# EPICS substitutions: LVREMOTE/LVREMOTE-IOC-01App/Db/lvremote_dds_tensile_stress_rig.substitutions
file lvremote_header.template {
    pattern { RECSIM, DISABLE }
    { "\$(RECSIM)", "\$(DISABLE)", }
}

file  lvremote_binary.template {
  pattern
    {DEVICE, P, NAME, IND, CONTROL, ZERO, ONE, VI, PORT, READONLY, DESCRIPTION, SCAN, HIGH}

    {"DDS_STRESS_RIG", "\$(P)", "ULIMIT:ENABLED", "EnableUL", "EnableUL", "False", "True", "C:/Instrument/Dev/ibex_vis/Drivers/DDS/dds Server.vi", "\$(NUM_PORT)", "", "Enable Upper Limit", "1 second", ""}
    {"DDS_STRESS_RIG", "\$(P)", "LLIMIT:ENABLED", "EnableLL", "EnableLL", "False", "True", "C:/Instrument/Dev/ibex_vis/Drivers/DDS/dds Server.vi", "\$(NUM_PORT)", "", "Enable Lower Limit", "1 second", ""}
    {"DDS_STRESS_RIG", "\$(P)", "SPEED:SET", "SetSpeed", "SetSpeed", "False", "True", "C:/Instrument/Dev/ibex_vis/Drivers/DDS/dds Server.vi", "\$(NUM_PORT)", "", "Set Speed", "1 second", "0.1"},
    {"DDS_STRESS_RIG", "\$(P)", "READ:START", "StartRead", "StartRead", "False", "True", "C:/Instrument/Dev/ibex_vis/Drivers/DDS/dds Server.vi", "\$(NUM_PORT)", "", "Start Reading", "1 second", "0.1"},
    {"DDS_STRESS_RIG", "\$(P)", "READ:STOP", "StopRead", "StopRead", "False", "True", "C:/Instrument/Dev/ibex_vis/Drivers/DDS/dds Server.vi", "\$(NUM_PORT)", "", "Stop Reading", "1 second", "0.1"},
    {"DDS_STRESS_RIG", "\$(P)", "MEAS:START", "StartMeasurement", "StartMeasurement", "False", "True", "C:/Instrument/Dev/ibex_vis/Drivers/DDS/dds Server.vi", "\$(NUM_PORT)", "", "Start Measurement", "1 second", "0.1"},
    {"DDS_STRESS_RIG", "\$(P)", "MEAS:STOP", "StopMeasurement", "StopMeasurement", "False", "True", "C:/Instrument/Dev/ibex_vis/Drivers/DDS/dds Server.vi", "\$(NUM_PORT)", "", "Stop Measurement", "1 second", "0.1"},
    {"DDS_STRESS_RIG", "\$(P)", "MOT:START", "StartMotor", "StartMotor", "False", "True", "C:/Instrument/Dev/ibex_vis/Drivers/DDS/dds Server.vi", "\$(NUM_PORT)", "", "Start Motor", "1 second", "0.1"},
    {"DDS_STRESS_RIG", "\$(P)", "MOT:STOP", "StopMotor", "StopMotor", "False", "True", "C:/Instrument/Dev/ibex_vis/Drivers/DDS/dds Server.vi", "\$(NUM_PORT)", "", "Stop Motor", "1 second", "0.1"}
}

file  lvremote_double.template {
  pattern
    {DEVICE, P, NAME, IND, CONTROL, VI, PORT, READONLY, WRITEONLY, SIMRECORD, DESCRIPTION, SCAN}

    {"DDS_STRESS_RIG", "\$(P)", "_SPEED", "Speed", "Speed", "C:/Instrument/Dev/ibex_vis/Drivers/DDS/dds Server.vi", "\$(NUM_PORT)", "","","", "Speed", "1 second"},
    {"DDS_STRESS_RIG", "\$(P)", "UPPER_LIMIT", "Upper Limit", "Upper Limit", "C:/Instrument/Dev/ibex_vis/Drivers/DDS/dds Server.vi", "\$(NUM_PORT)", "","","", "Upper Limit", "1 second"},
    {"DDS_STRESS_RIG", "\$(P)", "LOWER_LIMIT", "Lower Limit", "Lower Limit", "C:/Instrument/Dev/ibex_vis/Drivers/DDS/dds Server.vi", "\$(NUM_PORT)", "","","", "Lower Limit", "1 second"}
}

file  lvremote_enum.template {
  pattern
    {DEVICE, P, NAME, IND, CONTROL, VI, PORT, PORT2, READONLY, DESCRIPTION, SCAN, ZRST, ONST, TWST, THST,FRST,FVST,SXST, ZRVL, ONVL, TWVL, THVL,FRVL,FVVL,SXVL}

    {"DDS_STRESS_RIG", "\$(P)", "MODE:SPEED", "Mode", "Mode", "C:/Instrument/Dev/ibex_vis/Drivers/DDS/dds Server.vi", "\$(NUM_PORT)", "\$(STRING_PORT)", "", "Speed Mode", "1 second", "Manual", "Standard", "Load Const", "","","","", "0", "1", "2", "0","0","0","0"},
    {"DDS_STRESS_RIG", "\$(P)", "CONTROL:SPEED", "Control", "Control", "C:/Instrument/Dev/ibex_vis/Drivers/DDS/dds Server.vi", "\$(NUM_PORT)", "\$(STRING_PORT)", "", "Speed Control", "1 second", "Tacho", "Load", "Elongation", "Elongation 2","","","", "0", "1", "2", "3","0","0","0"},
    {"DDS_STRESS_RIG", "\$(P)", "DIRECTION:SPEED", "Direction", "Direction", "C:/Instrument/Dev/ibex_vis/Drivers/DDS/dds Server.vi", "\$(NUM_PORT)", "\$(STRING_PORT)", "", "Speed Direction", "1 second", "Forward", "Forward2", "Reverse", "","","","", "0", "1", "2", "3","0","0","0"},
    {"DDS_STRESS_RIG", "\$(P)", "MODE:STAT", "Mode String", "Set Mode", "C:/Instrument/Dev/ibex_vis/Drivers/DDS/dds Server.vi", "\$(NUM_PORT)", "\$(STRING_PORT)", "", "Set Mode", "1 second", "Manual", "Standard", "Load Const", "Elong 2","","","", "0", "1", "2", "3","0","0","0"},
    {"DDS_STRESS_RIG", "\$(P)", "MOT:MODE", "Motor Control Mode String", "Set Control", "C:/Instrument/Dev/ibex_vis/Drivers/DDS/dds Server.vi", "\$(NUM_PORT)", "\$(STRING_PORT)", "", "Set Control", "1 second", "Tacho", "Load", "Elongation", "Elongation 2","","","", "0", "1", "2", "3","0","0","0"},
    {"DDS_STRESS_RIG", "\$(P)", "DIR", "Direction String", "Set Direction", "C:/Instrument/Dev/ibex_vis/Drivers/DDS/dds Server.vi", "\$(NUM_PORT)", "\$(STRING_PORT)", "", "Set Direction", "1 second", "Forward", "Forward2", "Reverse", "","","","", "0", "1", "2", "3","0","0","0"},
    {"DDS_STRESS_RIG", "\$(P)", "CHANNEL", "Choose Channel", "Choose Channel", "C:/Instrument/Dev/ibex_vis/Drivers/DDS/dds Server.vi", "\$(NUM_PORT)", "\$(STRING_PORT)", "", "Channel", "1 second", "Time", "Load", "Elongation", "Elong2","","","", "0", "1", "2", "3","0","0","0"}

    {"DDS_STRESS_RIG", "\$(P)", "MOT:STAT", "Motor Status String", "Motor Status String", "C:/Instrument/Dev/ibex_vis/Drivers/DDS/dds Server.vi", "\$(NUM_PORT)", "\$(STRING_PORT)", "#", "Motor Status", "1 second", "Stop", "Forward", "Reverse", "","","","", "0", "1", "2", "0","0","0","0"},
    {"DDS_STRESS_RIG", "\$(P)", "CON:STAT", "Control Status String", "Control Status String", "C:/Instrument/Dev/ibex_vis/Drivers/DDS/dds Server.vi", "\$(NUM_PORT)", "\$(STRING_PORT)", "#", "Control Status", "1 second", "Idle", "Read", "Active","Hold","HoldEnd","AutoZero","AutoKeepConst", "0","1","2","3","4","5","6"},
    {"DDS_STRESS_RIG", "\$(P)", "TEMP:STAT", "Temp Status String", "Temp Status String", "C:/Instrument/Dev/ibex_vis/Drivers/DDS/dds Server.vi", "\$(NUM_PORT)", "\$(STRING_PORT)", "#", "Temp Status String", "1 second", "Stop", "Heating", "Cooling", "","","","", "0", "1", "2", "0","0","0","0"},
}

file lvremote_array.template {
  pattern
  {DEVICE, P, NAME, IND, CONTROL, VI, PORT, DESCRIPTION, SCAN, TYPE, INDEX}

  {"DDS_STRESS_RIG", "\$(P)", "ARRAY", "Display", "Display", "C:/Instrument/Dev/ibex_vis/Drivers/DDS/dds Server.vi", "\$(NUM_PORT)", "Display", "1 second", "DOUBLE", "7"}
}
